//Placeholder, WIP --> need to define what purpose this struct serves
TYPE ST_SegmentNumber :
STRUCT
    refIn: REFERENCE TO ST_SegmentNumberIn;
    refOut: REFERENCE TO ST_SegmentNumberOut;
END_STRUCT
END_TYPE

(* stored: Version 1.1.0.1
   DUT ST_SegmentNumber: Id {12f01272-bde2-0fa6-0a62-97eed6c2e8c3} *)
